(* CoDeSys 2.3 export: IED_STATE_EN_INIT.EXP *)

(* POU IED_STATE_EN_INIT, ST *)
FUNCTION_BLOCK IED_STATE_EN_INIT
VAR_INPUT
	IED_STATE: INT;
END_VAR
VAR_OUTPUT
	IED_STATE_CTS: BOOL;
END_VAR
VAR
	previous_state: INT;
END_VAR
IF IED_STATE <> previous_state
	THEN IED_STATE_CTS := TRUE;
	ELSE IED_STATE_CTS := FALSE;
END_IF

previous_state := IED_STATE;
END_FUNCTION_BLOCK
